{attribute 'linkalways'} 
{attribute 'no_explicit_call' := 'This FB is a CLASS and must be accessed using methods or properties'}
{attribute 'enable_dynamic_creation'}
FUNCTION_BLOCK _ETcVnContainerExportFormat EXTENDS EnumDatatypeBase
VAR
	localData : ETcVnContainerExportFormat;
	activeData : REFERENCE TO ETcVnContainerExportFormat;
	enumBaseDatatype : _UINT(localData);
END_VAR

METHOD PRIVATE AddLocalEnumeration
VAR_INPUT
	Enumeration : T_MAXSTRING;
	Value : ETcVnContainerExportFormat;
END_VAR
AddEnumeration(Enumeration, Value);
END_METHOD

PROPERTY PUBLIC Address : PVOID
GET
Address := ADR(activeData);
END_GET
END_PROPERTY

METHOD PUBLIC ClearReference
VAR_INPUT
END_VAR
activeData REF= localData;
SetBaseDatatypeReference();
END_METHOD

METHOD PUBLIC Clone : I_Datatype
VAR
    pClone : POINTER TO _ETcVnContainerExportFormat;
END_VAR
pClone := __NEW(_ETcVnContainerExportFormat(InitialValue := Value));
Clone := pClone^;
END_METHOD

METHOD FB_init : BOOL
VAR_INPUT
	bInitRetains : BOOL; // if TRUE, the retain variables are initialized (warm start / cold start)
	bInCopyCode : BOOL;  // if TRUE, the instance afterwards gets moved into the copy code (online change)
	InitialValue : ETcVnContainerExportFormat;
END_VAR
localData := InitialValue;
AddBaseDatatype(enumBaseDatatype);
ClearReference();

AddLocalEnumeration('TCVN_CEF_XML', ETcVnContainerExportFormat.TCVN_CEF_XML);
AddLocalEnumeration('TCVN_CEF_XML_SERIALIZED', ETcVnContainerExportFormat.TCVN_CEF_XML_SERIALIZED);
AddLocalEnumeration('TCVN_CEF_CSV', ETcVnContainerExportFormat.TCVN_CEF_CSV);
AddLocalEnumeration('TCVN_CEF_BINARY', ETcVnContainerExportFormat.TCVN_CEF_BINARY);
END_METHOD

PROPERTY PUBLIC Identifier : T_MAXSTRING
GET
Identifier := 'ETcVnContainerExportFormat';
END_GET
END_PROPERTY

METHOD IsEnumeratorValueEqual : BOOL
VAR_INPUT
	Enumerator : I_KeyValueForwardEnumerator;
END_VAR
VAR
	storedValue : ETcVnContainerExportFormat;
END_VAR
IF NOT Enumerator.TryGet(storedValue) THEN
	RETURN;
END_IF

IsEnumeratorValueEqual := storedValue = activeData;
END_METHOD

METHOD PUBLIC MakeReferenceTo
VAR_INPUT
	ReferenceTarget : REFERENCE TO ETcVnContainerExportFormat;
END_VAR
activeData REF= ReferenceTarget;
SetBaseDatatypeReference();
END_METHOD

METHOD PROTECTED SetBaseDatatypeReference
VAR_INPUT
END_VAR
enumBaseDatatype.MakeReferenceTo(activeData);
END_METHOD

PROPERTY PUBLIC Size : UDINT
GET
Size := SIZEOF(activeData);
END_GET
END_PROPERTY

METHOD TryMakeReferenceTo : BOOL
VAR_INPUT
	Target : I_Datatype;
END_VAR
VAR
	targetAsEnum : I_EnumDatatype;
	pTargetData : POINTER TO ETcVnContainerExportFormat;
END_VAR
IF NOT Target.TryResolveAsEnumDatatype(targetAsEnum) THEN
	RETURN;
END_IF

IF targetAsEnum.Identifier <> Identifier THEN
	RETURN;
END_IF

pTargetData := Target.Address;
activeData REF= pTargetData^;
SetBaseDatatypeReference();
TryMakeReferenceTo := TRUE;
END_METHOD

PROPERTY PUBLIC Value : ETcVnContainerExportFormat
GET
Value := activeData;
END_GET
SET
activeData := Value;
END_SET
END_PROPERTY

END_FUNCTION_BLOCK

(* stored: Version 1.1.0.1, ProductVersion 3.1.4024.12
   POU _ETcVnContainerExportFormat: Id {8c1a2ac2-0b77-4ffd-9ae0-e40f64b06cff}, SpecialFunc None
   Folder Constructor: Id {ca294c03-6ab4-4d22-940a-d00702a34493}
   Folder Private: Id {3da26f00-2972-43e8-ae5e-0b7d8b4103af}
   Folder Protected: Id {f7b69b1e-89ba-4361-9cd8-2ff98ebba763}
   Method AddLocalEnumeration: Id {d3dcf010-33eb-412f-84a0-d46fac9e8acf}
   Property Address: Id {fdbcc058-093b-41e6-8019-a73b64d09c86}
   Get Get: Id {7a5e3db2-c097-42bc-acc5-4a258c30a385}
   Method ClearReference: Id {0a675f20-93a4-4f5f-86d4-07b16680b01c}
   Method Clone: Id {7b6e66f0-677e-4c5d-9526-33b446e4b8e7}
   Method FB_init: Id {2943c004-53a5-4ae4-ab93-4c016a37ef0d}
   Property Identifier: Id {457ea0d1-53f1-41e9-8408-175a00a1591f}
   Get Get: Id {dc049d7b-8e61-47be-aaa4-e56d6d40638e}
   Method IsEnumeratorValueEqual: Id {d50af9ad-a714-4dff-aca2-756987a3e430}
   Method MakeReferenceTo: Id {a799a51f-da13-40d0-baaa-9b5fd6b2e3b2}
   Method SetBaseDatatypeReference: Id {e9559187-8a35-4da8-bdd1-ca23d4731d17}
   Property Size: Id {ed303e1c-a4bc-468d-bb78-df9ff76209c4}
   Get Get: Id {03e04bcb-c335-4010-bdc1-305b838868ed}
   Method TryMakeReferenceTo: Id {075afda8-fcbd-4e80-89a9-5173a80c27d7}
   Property Value: Id {38ca7cde-8ed4-4707-b172-028d5c65d4c8}
   Get Get: Id {a5d8eaf8-996b-46c2-8d14-7f02e44bf5cf}
   Set Set: Id {62d96a55-bc20-4871-bd5e-7227b2125ead} *)
